Staubli VAL3: CartesianForce.pjx

--- CartesianForce.pjx ---
Parameters version=s7.9.1 stackSize=5000 millimeterUnit=true
Data file=CartesianForce.dtx

--- CartesianForce.dtx ---
public num fx
public num fy
public num fz
public num frx
public num fry
public num frz
